FUNCTION F_LowestReal : REAL
VAR_INPUT
	Value1																: REAL;
	Value2																: REAL;
END_VAR
VAR
END_VAR

// F_LowestReal
// Rev 1.0 - March 14, 2024

F_LowestReal															:= SEL(Value1 < Value2, Value2, Value1);

END_FUNCTION

(* stored: Version 1.1.0.1, ProductVersion 3.1.4024.12
   POU F_LowestReal: Id {06eaf0f5-fdf3-4de8-b4e4-1f9fb6ec5ab4}, SpecialFunc None *)
